FUNCTION_BLOCK FB_InfeedConveyor
VAR_INPUT
    iMotor          : I_Drive;
    iProductCam     : I_DigitalSensor;
    
    // --- NEW: Commands from Main Machine ---
    bEnable         : BOOL; // <--- ADD THIS LINE
    
    // --- Machine Parameters ---
    fTargetVelocity : LREAL := 100.0;
END_VAR
VAR
END_VAR

// The conveyor is very simple for now. 
// It just ensures the motor is enabled and running.
IF iMotor <> 0 THEN
    iMotor.P_Enabled := bEnable;
    
    // ADDED: The required nDirection parameter to satisfy the interface
    iMotor.M_MoveVelocity(fVelocity := fTargetVelocity, nDirection := 1);
END_IF

END_FUNCTION_BLOCK

(* stored: Version 1.1.0.1
   POU FB_InfeedConveyor: Id {bd972d02-828a-4a6c-9ef5-f96cad8432c6}, SpecialFunc None *)
